FUNCTION_BLOCK AxisController
VAR_INPUT
	bExecute: BOOL;
	fSpeed : LREAL := 360;
END_VAR
VAR
	mcReset			: MC_Reset;
	mcPower			: MC_Power;
	mcMoveVelo		: MC_MoveVelocity;
	mcStop			: MC_Stop;
	
	iState: UINT;;
END_VAR
VAR_IN_OUT
	Axis : AXIS_REF;
END_VAR
VAR_OUTPUT
	bDone : BOOL;
END_VAR

mcReset(Axis:=Axis);
mcReset.Execute := FALSE;

mcPower(Axis:=Axis, Enable:=TRUE, Enable_Positive:=TRUE, Enable_Negative:=TRUE);

mcMoveVelo(Axis:=Axis);
mcMoveVelo.Execute := FALSE;

CASE iState OF
	0:		
		IF bExecute THEN
			iState:= 10;
		END_IF
		
	10: 
		// Reset the axis
		mcReset.Execute:=TRUE;
		iState := 20;
		bDone:= FALSE;
	
	20: 
		// Wait for reset to complete
		IF McReset.Done THEN
			iState := 30;
		ELSIF McReset.Error THEN
			iState := 999;
		END_IF
	
	30:
		// Set the power!
		IF McPower.Status THEN
			iState := 40;
		END_IF
		
	40: 
		// Move at constant velo
		mcMoveVelo.Execute := TRUE;
		mcMoveVelo.Velocity:=fSpeed;
		
		iState:= 50;
	
	50: 
		// Done.
		IF mcMoveVelo.InVelocity THEN
			bDone := TRUE;
			iState := 0;
		END_IF
		
END_CASE

END_FUNCTION_BLOCK

(* stored: Version 1.1.0.1, ProductVersion 3.1.4022.10
   POU AxisController: Id {03a3ed9a-8b31-4918-82ec-f19698baf36a}, SpecialFunc None *)
